FUNCTION_BLOCK FB_CheckTasks
VAR_INPUT
	tTimeTaskError: BOOL;
END_VAR
VAR_OUTPUT
END_VAR
VAR
	i: UINT;
	tAreAllTasksComeplete: BOOL;
	tSumTaskTime: LREAL;
	tTaskTimeError: BOOL;
END_VAR
VAR_IN_OUT
	iqPartData:typeStation; //insert station data
END_VAR
















//theme:MPa8jVeIbTM

//check all tasks for depth or skipped

//set complete logic
tAreAllTasksComeplete:=TRUE;
tSumTaskTime:=0.0;



//scan status of current tasks and inverse logic TRUE if the task is completed
FOR i := 1 TO maxNumTasks DO;
	
	IF  NOT iqPartData.part.tasks[i].IsTaskEnabled THEN
		tAreAllTasksComeplete := FALSE;
	END_IF
	
	IF  NOT iqPartData.part.tasks[i].IsTaskComplete THEN
		tAreAllTasksComeplete := FALSE;
	END_IF
	
	IF  iqPartData.part.tasks[i].IsTaskEnabled THEN
		//get summation of cycle time from tasks
		tSumTaskTime := tSumTaskTime + iqPartData.part.tasks[i].CycleTimeActual;
	END_IF
	
END_FOR

//if the loop did not detect and tasks not enabled, or tasks not complete,
//then set the station complete to TRUE
IF tAreAllTasksComeplete THEN
	iqPartData.part.PartComplete:=TRUE;
	ELSE
	//do not reset here, PartComplete resets when part removed via gantry/conveyor
END_IF


//check if sum of task cycle time does not match station declared station time
IF tSumTaskTime = iqPartData.part.CycleTimeTarget THEN //compare reals??1?
	tTaskTimeError:=TRUE;
	ELSE
	tTimeTaskError:=FALSE;
END_IF

END_FUNCTION_BLOCK

(* stored: Version 1.1.0.1, ProductVersion 3.1.4024.12
   POU FB_CheckTasks: Id {c4783f8d-b6d2-4c4f-98af-16aaa73e252f}, SpecialFunc None *)
